{attribute 'qualified_only'}
{attribute 'strict'}

//-----------------------------------------------------------------------------------------
//
//                  				ENUM_User_Level
//
//							Enumération des niveaux d'utilisateurs			
//-----------------------------------------------------------------------------------------
//
//Auteur: G.GOETZ
//Création: 04.03.2026
//Dernière modification : 04.03.2026 (G.GOETZ)
//       			
//-----------------------------------------------------------------------------------------
//
//     							Liste des modifications  	
//
// 04.03.2026 (G.GOETZ) -> Création		
//-----------------------------------------------------------------------------------------

TYPE ENUM_User_Level :
(
	None := 0 ,
	Admin := 1 ,
	Maintenance := 2 ,
	Operator := 3 
);
END_TYPE

(* stored: Version 1.1.0.1, ProductVersion 3.1.4026.17
   DUT ENUM_User_Level: Id {0f672b10-f6c2-4864-b9e3-7ffd39b959b9} *)
